RoboDK station: wlkata_demo.rdk

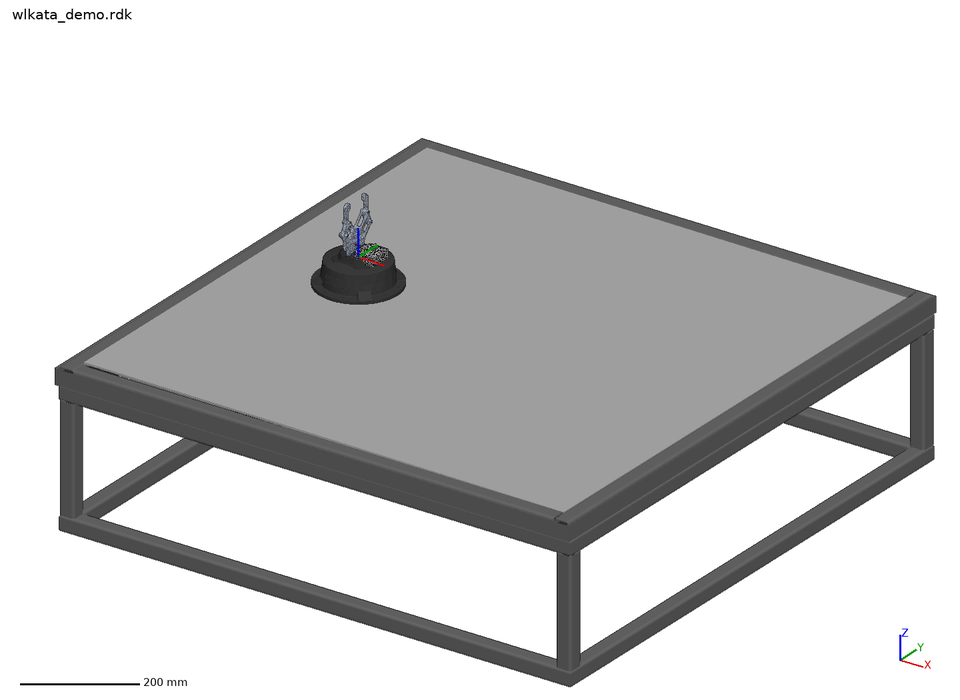
[picture v0: the station drawn from its stored meshes, robots at their saved joint values, targets as dots, program paths as lines]
Station wlkata_demo (saved by RoboDK 5.5.2). Poses are relative to the parent item; angles as X-Y-Z fixed-axis rotations.
  - object Table 108x114x32in at (0, 0, 0) mm, size 1051.6 x 1071.9 x 311.4 mm, geometry from Table-108x114x32in.sld
  - frame base-frame at (239.05, 9.81, 360) mm, rotated rx 0 ry 0 rz -1.06 deg
    - robot robot-wlkata (model Wlkata Mirobot): 6 axes, payload 0.4 kg, reach 315 mm, repeatability 0.2 mm, weight 1.5 kg
        joint limits [-100, -60, -180, -180, -180, -180] to [100, 90, 50, 180, 50, 180]; home [0, 0, 0, 0, 0, 0]; saved at [-30.373, 16.472, 26.663, -5.469, -72.702, -38.24]
      - tool servo-gripper, TCP at (0, 0, 0) mm, size 78 x 62.4 x 128.4 mm, geometry from Gripper.IGS
